// Mitsubishi GX Works2 project: 0319_인터로크2   PLC: Q03UDV

PROGRAM MAIN
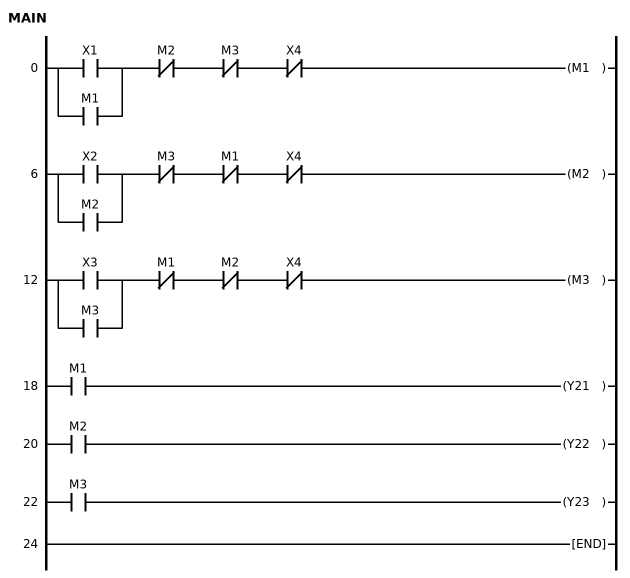
0     LD      X1
      OR      M1
      ANI     M2
      ANI     M3
      ANI     X4
      OUT     M1
6     LD      X2
      OR      M2
      ANI     M3
      ANI     M1
      ANI     X4
      OUT     M2
12    LD      X3
      OR      M3
      ANI     M1
      ANI     M2
      ANI     X4
      OUT     M3
18    LD      M1
      OUT     Y21
20    LD      M2
      OUT     Y22
22    LD      M3
      OUT     Y23
24    END
END_PROGRAM
